FUNCTION_BLOCK FUNCTION
  {SET_ATTRIBUTE(OpcUa, SERVICE)}
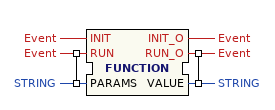
  EVENT_INPUT
    INIT;
    RUN WITH PARAMS;
  END_EVENT
  EVENT_OUTPUT
    INIT_O;
    RUN_O WITH VALUE;
  END_EVENT
  VAR_INPUT
    PARAMS : STRING; {SET_ATTRIBUTE(OpcUa, Variable)}
  END_VAR
  VAR_OUTPUT
    VALUE : STRING; {SET_ATTRIBUTE(OpcUa, Variable)}
  END_VAR
END_FUNCTION_BLOCK
